RoboDK station: Piles.rdk

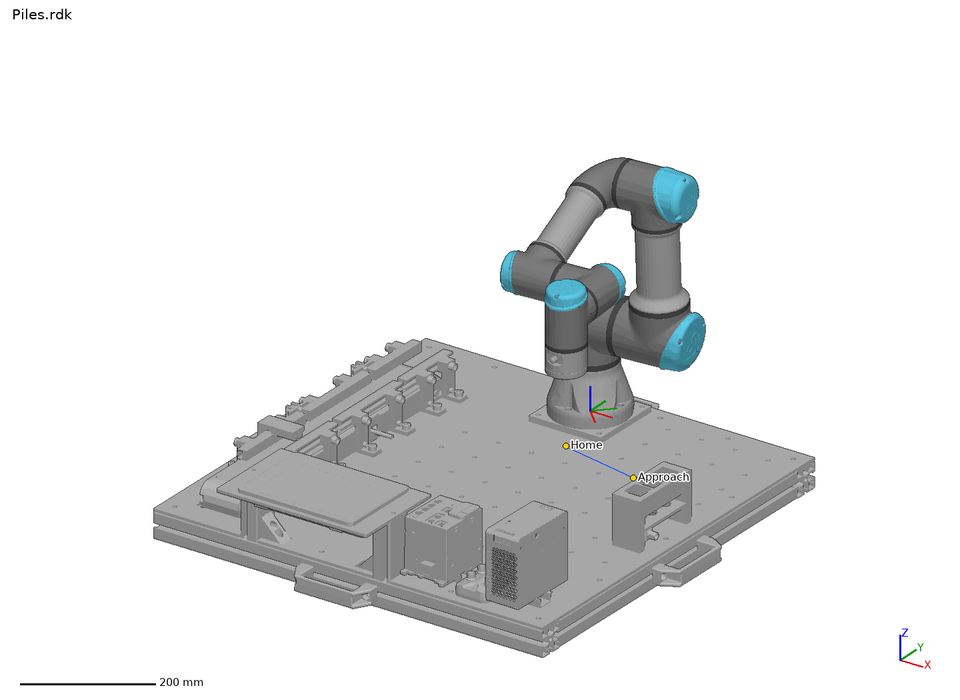
[picture v0: the station drawn from its stored meshes, robots at their saved joint values, targets as dots, program paths as lines]
Station Piles (saved by RoboDK 5.3.0). Poses are relative to the parent item; angles as X-Y-Z fixed-axis rotations.
  - frame UR3e Base at (0, 0, 0) mm, rotated rx 0 ry 0 rz -45 deg
    - robot UR3e: 6 axes, payload 3 kg, reach 500 mm, repeatability 0.03 mm, weight 11 kg
        modified DH rows (alpha deg, a mm, theta deg, d mm): 0, 0, 0, 151.9; 90, 0, 180, 0; 0, 243.55, 0, 0; 0, 213.2, 0, 131.05; -90, 0, 0, 85.35; 90, 0, 180, 92.1
        joint limits [-360, -360, -360, -360, -360, -360] to [360, 360, 360, 360, 360, 360]; home [0, -90, -90, 0, 90, 0]; saved at [139.875, 273.237, -251.461, -111.776, 270, 4.875]
      - tool Tool 1, TCP at (0, 0, 124.6) mm
  - frame CAD at (0, 0, 0) mm
    - object MiniCellule_Rev3 at (349, -599, -37.5) mm, rotated rx 0 ry -90 rz 0 deg, size 184.2 x 802 x 782 mm, geometry from MiniCellule_Rev3.stp
    - target Home (Cartesian target) at (155.82, -284.88, 99.27) mm, rotated rx 180 ry 0 rz -180 deg; joints [139.875, 273.237, -251.461, -111.776, 270, 4.875] of UR3e
    - target Approach (Cartesian target) at (299.64, -316.39, 100.08) mm, rotated rx 180 ry 0 rz -180 deg; joints [160.94, 299.207, -306.67, -82.537, 270, 25.94] of UR3e
  - program Prog1 (4 instructions, listed below)

--- program Prog1 (robot UR3e) ---
  Définir Ref.: CAD
  Choisir Outil: Tool 1
  MoveJ (Home)
  MoveJ (Approach)
